# B&R Automation Studio project lab4
Automation Studio 4.5.2.102

## Configuration Real

### Hardware
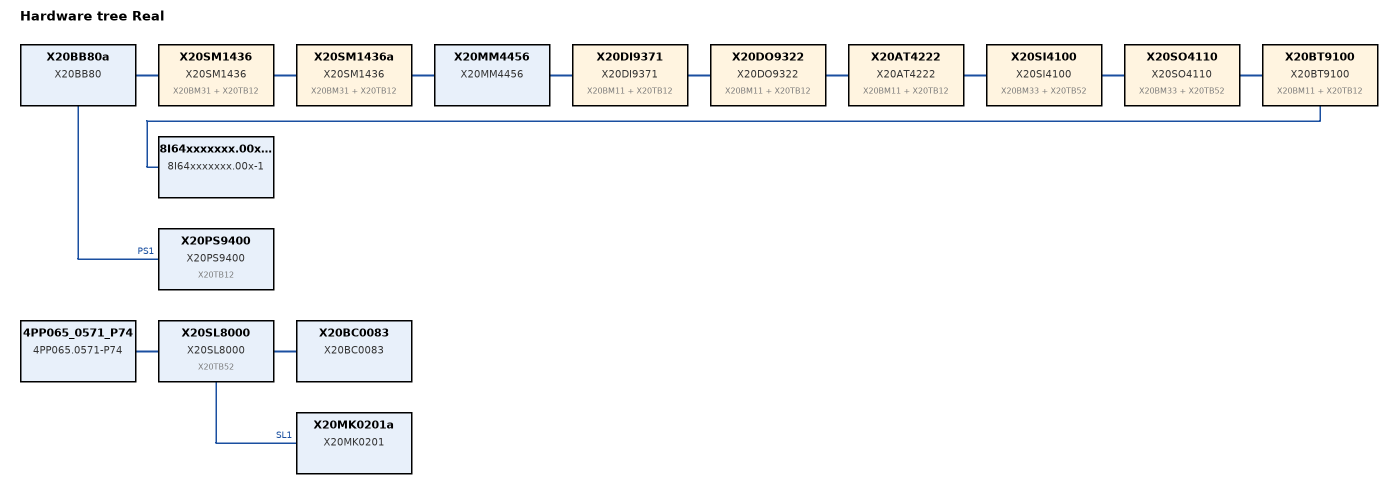
```
4PP065_0571_P74 : 4PP065.0571-P74 v1.1.2.0
  Connector IF5:
    ActivateDevice = 1
    Mode = Manual
    InternetAddress = 10.0.1.10
    SubnetMask = 255.255.255.0
  ConfigurationID = LabBR
  TimerDeviceType = EPLX2X
  TimerDevice = 4PP065_0571_P74.IF4
  TaskClassIdleTime = 2000
  Cyclic1Duration = 2000
  Cyclic1Tolerance = 0
  Cyclic1Output = 1
  Cyclic3Tolerance = 0
  VcObjectName = Visu
8I64xxxxxxx.00x-1 : 8I64xxxxxxx.00x-1 v1.3.9.1  [X2X1 -> X20BT9100.X2X1 [Cable Type=X2XCable, Length=10, Version=1.0.0.2]]
  BothEndSwitchesAreNormallyOpen_r1 = on
  QuickStopIsNormallyOpen_r1 = on
X20AT4222 : X20AT4222 v1.2.3.0  [SS1 -> X20TB12f.SS; SL -> X20BM11c.SL1]
X20BB80a : X20BB80 v1.0.2.0
X20BC0083 : X20BC0083 v2.7.0.0  [PLK1 -> X20SL8000.PLK2 (NodeNumber=2) [Cable Type=PowerlinkCable, Length=10, Version=1.0.0.2]; SL -> X20BB80a.SL1]
X20BM11a : X20BM11 v1.0.0.1  [X2X1 -> X20MM4456.X2X2]
X20BM11b : X20BM11 v1.0.0.1  [X2X1 -> X20BM11a.X2X2]
X20BM11c : X20BM11 v1.0.0.1  [X2X1 -> X20BM11b.X2X2]
X20BM11d : X20BM11 v1.0.0.1  [X2X1 -> X20BM33b.X2X2]
X20BM31a : X20BM31 v1.0.0.1  [X2X1 -> X20BB80a.IF1]
X20BM31b : X20BM31 v1.0.0.1  [X2X1 -> X20BM31a.X2X2]
X20BM33a : X20BM33 v1.0.0.4  [X2X1 -> X20BM11c.X2X2]
X20BM33b : X20BM33 v1.0.0.4  [X2X1 -> X20BM33a.X2X2]
X20BT9100 : X20BT9100 v1.0.3.0  [SS1 -> X20TB12g.SS; SL -> X20BM11d.SL1]
X20DI9371 : X20DI9371 v1.0.2.0  [SS1 -> X20TB12d.SS; SL -> X20BM11a.SL1]
X20DO9322 : X20DO9322 v1.0.3.0  [SS1 -> X20TB12e.SS; SL -> X20BM11b.SL1]
X20MK0201a : X20MK0201 v1.0.0.0  [SL -> X20SL8000.SL1]
X20MM4456 : X20MM4456 v1.1.5.0  [X2X1 -> X20BM31b.X2X2]
X20PS9400 : X20PS9400 v1.0.2.4  [SS1 -> X20TB12b.SS; PS -> X20BB80a.PS1]
X20SI4100 : X20SI4100 v1.10.1.1  [SS1 -> X20TB52b.SS; SL -> X20BM33a.SL1]
X20SL8000 : X20SL8000 v1.6.5.1  [PLK1 -> 4PP065_0571_P74.IF4 (NodeNumber=1) [Cable Type=PowerlinkCable, Length=10, Version=1.0.0.2]; PLK2 -> X20BC0083.PLK1 (NodeNumber=1) [Cable Type=PowerlinkCable, Length=10, Version=1.0.0.2]; SS1 -> X20TB52a.SS]
  SafeProject = SafeLOGIC-1
X20SM1436 : X20SM1436 v1.4.2.1  [SS1 -> X20TB12a.SS; SL -> X20BM31a.SL1]
X20SM1436a : X20SM1436 v1.4.2.1  [SS1 -> X20TB12c.SS; SL -> X20BM31b.SL1]
X20SO4110 : X20SO4110 v1.10.1.1  [SS1 -> X20TB52c.SS; SL -> X20BM33b.SL1]
  SafeLogicID = 2
  SafeModuleID = 3
X20TB12a : X20TB12 v1.0.0.0
X20TB12b : X20TB12 v1.0.0.0
X20TB12c : X20TB12 v1.0.0.0
X20TB12d : X20TB12 v1.0.0.0
X20TB12e : X20TB12 v1.0.0.0
X20TB12f : X20TB12 v1.0.0.0
X20TB12g : X20TB12 v1.0.0.0
X20TB52a : X20TB52 v1.0.0.1
X20TB52b : X20TB52 v1.0.0.1
X20TB52c : X20TB52 v1.0.0.1
```

### IoMap.iom - 4PP065_0571_P74/IoMap.iom
```iecst
VAR_CONFIG
	::SDCAxisCt2:posEnable.enable AT %IX."X20DI9371".DigitalInput04; (*Insert your comment here...*)
	::SDCAxisCt2:posEnableRight.enable AT %IX."X20DI9371".DigitalInput05; (*Insert your comment here...*)
	::SDCAxisCt1:posEnable.enable AT %IX."X20DI9371".DigitalInput04; (*Insert your comment here...*)
	::SDCAxisCt1:posEnableRight.enable AT %IX."X20DI9371".DigitalInput05; (*Insert your comment here...*)
	::SDCAxisCtr:posEnable.enable AT %IX."X20DI9371".DigitalInput02; (*Insert your comment here...*)
	::SDCAxisCtr:posEnableRight.enable AT %IX."X20DI9371".DigitalInput03; (*Insert your comment here...*)
	Cyclic#1.gAxis03_DrvIf.iLifeCnt AT %IB."8I64xxxxxxx.00x-1".SDC_LifeCnt;
	Cyclic#1.gAxis03_DrvIf.iDrvOK AT %IX."8I64xxxxxxx.00x-1".ETAD_Input_Bool_02;
	Cyclic#1.gAxis03_DrvIf.oSetTime AT %QW."8I64xxxxxxx.00x-1".SDC_SetTime;
	Cyclic#1.gAxis03_DrvIf.oSetPos AT %QW."8I64xxxxxxx.00x-1".LFRD_Output;
	Cyclic#1.gAxis03_DiDoIf.iLifeCntDriveReady AT %IB."8I64xxxxxxx.00x-1".SDC_LifeCnt;
	Cyclic#1.gAxis03_DiDoIf.iLifeCntDriveEnable AT %IB."8I64xxxxxxx.00x-1".SDC_LifeCnt;
	Cyclic#1.gAxis03_DiDoIf.oDriveEnable AT %QX."8I64xxxxxxx.00x-1".CMDD_Output_Bool_00;
	Cyclic#1.gAxis03_ModuleOk AT %QX."8I64xxxxxxx.00x-1".CMDD_Output_Bool_01;
	Cyclic#1.gAxis03_ModuleOk AT %QX."8I64xxxxxxx.00x-1".CMDD_Output_Bool_02;
	Cyclic#1.gAxis03_ModuleOk AT %IX."8I64xxxxxxx.00x-1".ModuleOk;
	Cyclic#1.gAxis03_DiDoIf.oDriveEnable AT %QX."8I64xxxxxxx.00x-1".CMDD_Output_Bool_03;
	Cyclic#1.gAxis03_DiDoIf.iDriveReady AT %IX."8I64xxxxxxx.00x-1".ETAD_Input_Bool_02;
	::SDCAxisCtr:pwm_period AT %QW."X20MM4456".PeriodDurationPWM;
	::SDCAxisCtr:coil_pwm_value AT %QW."X20MM4456".PulseWidthCurrentPWM04;
	::SDCAxisCtr:axis_X.pwm_value AT %QW."X20MM4456".PulseWidthCurrentPWM01;
	::SDCAxisCtr:axis_X.reset_error AT %QX."X20MM4456".ClearError01;
	::SDCAxisCtr:axis_X.reset_counter AT %QX."X20MM4456".ResetCounter01;
	::SDCAxisCtr:axis_X.counter AT %IW."X20MM4456".Counter01;
	::SDCAxisCtr:axis_X.endswitch_a_reached AT %IX."X20MM4456".StatusInput03; (*Logical condition input 01=Motor 01:A*)
	::SDCAxisCtr:axis_X.endswitch_b_reached AT %IX."X20MM4456".StatusInput04; (*Logical condition input 02=Motor 01:B*)
	::SDCAxisCtr:coil_powered AT %IX."X20DI9371".DigitalInput01;
	::SDCAxisCt1:axis_Y.pwm_value AT %QW."X20MM4456".PulseWidthCurrentPWM02;
	::SDCAxisCt1:axis_Y.reset_error AT %QX."X20MM4456".ClearError02;
	::SDCAxisCt1:axis_Y.reset_counter AT %QX."X20MM4456".ResetCounter02;
	::SDCAxisCt1:axis_Y.counter AT %IW."X20MM4456".Counter02;
	::SDCAxisCt1:axis_Y.endswitch_a_reached AT %IX."X20MM4456".StatusInput07;
	::SDCAxisCt1:axis_Y.endswitch_b_reached AT %IX."X20MM4456".StatusInput08;
	::SDCAxisCt2:axis_Z.pwm_value AT %QW."X20MM4456".PulseWidthCurrentPWM03;
	::SDCAxisCt2:axis_Z.reset_error AT %QX."X20MM4456".ClearError03;
	::SDCAxisCt2:axis_Z.reset_counter AT %QX."X20MM4456".ResetCounter03;
	::SDCAxisCt2:axis_Z.counter AT %IW."X20MM4456".Counter03;
	::SDCAxisCt2:axis_Z.endswitch_a_reached AT %IX."X20MM4456".StatusInput11;
	::SDCAxisCt2:axis_Z.endswitch_b_reached AT %IX."X20MM4456".StatusInput12;
	::SDCAxisCt1:coil_powered AT %IX."X20DI9371".DigitalInput02;
	::SDCAxisCt2:coil_powered AT %IX."X20DI9371".DigitalInput03;
END_VAR
```

### Acp10map1.ncm - 4PP065_0571_P74/Motion/Acp10map1.ncm
```
NcMapping (NcSwId=ACP10, DisabledNodesAreHidden=False)
  NcObject AxisX (ModuleAddress=SDC_IF1.ST2, InterfaceType=SDC, Type=ncAXIS, Channel=1, AcoposSimulation=Off, InitParameter=AxisInit, AcoposParameter=AxisApt, AdditionalData=CNC_Enabled="1" , Disabled=FALSE, ModuleDisabled=FALSE)
  NcObject AxisY (ModuleAddress=SDC_IF1.ST3, InterfaceType=SDC, Type=ncAXIS, Channel=1, AcoposSimulation=Off, InitParameter=AxisInit, AcoposParameter=AxisApt, AdditionalData=CNC_Enabled="1" , Disabled=FALSE)
  NcObject AxisZ (ModuleAddress=SDC_IF1.ST4, InterfaceType=SDC, Type=ncAXIS, Channel=1, AcoposSimulation=Off, InitParameter=AxisInit, AcoposParameter=AxisApt, AdditionalData=CNC_Enabled="1" , Disabled=FALSE)
```

## Logical view

### Package Logical/Libraries - Global libraries

### Library Logical/Libraries/Library (ANSIC)

#### Library.fun
```iecst
FUNCTION_BLOCK FB_Motor (*TODO: Add your comment here*) (*$GROUP=User,$CAT=User,$GROUPICON=User.png,$CATICON=User.png*)
	VAR_INPUT
		in : REAL;
	END_VAR
	VAR_OUTPUT
		out_w : REAL;
		out_phi : REAL;
	END_VAR
	VAR
		k_e : REAL;
		T_m : REAL;
		dt : REAL;
		integrator : FB_Integrator;
		integrator_phi : FB_Integrator;
	END_VAR
END_FUNCTION_BLOCK

FUNCTION_BLOCK FB_Integrator (*TODO: Add your comment here*) (*$GROUP=User,$CAT=User,$GROUPICON=User.png,$CATICON=User.png*)
	VAR_INPUT
		in : REAL;
		dt : REAL;
	END_VAR
	VAR_OUTPUT
		out : REAL;
	END_VAR
	VAR
		state : REAL := 0.0;
	END_VAR
END_FUNCTION_BLOCK

FUNCTION_BLOCK FB_Controller (* *) (*$GROUP=User,$CAT=User,$GROUPICON=User.png,$CATICON=User.png*)
	VAR_INPUT
		in : REAL;
	END_VAR
	VAR_OUTPUT
		out : REAL;
	END_VAR
	VAR
		k_i : REAL;
		sum : REAL;
		k_p : REAL;
		dt : REAL;
		max_abs_value : REAL;
		integrator : FB_Integrator;
		last_sum : REAL;
	END_VAR
END_FUNCTION_BLOCK

FUNCTION_BLOCK FB_Endswitch (*TODO: Add your comment here*) (*$GROUP=User,$CAT=User,$GROUPICON=User.png,$CATICON=User.png*)
	VAR_INPUT
		in : REAL;
		neg_value : REAL;
		pos_value : REAL;
	END_VAR
	VAR_OUTPUT
		neg_reached : BOOL;
		pos_reached : BOOL;
	END_VAR
END_FUNCTION_BLOCK

FUNCTION_BLOCK FB_Axis (*TODO: Add your comment here*) (*$GROUP=User,$CAT=User,$GROUPICON=User.png,$CATICON=User.png*)
	VAR_INPUT
		reset_error : BOOL;
		endswitch_a_reached : BOOL;
		endswitch_b_reached : BOOL;
		pwm_percentage : SINT;
	END_VAR
	VAR_OUTPUT
		reset_counter : BOOL;
		pwm_value : INT;
	END_VAR
	VAR_OUTPUT RETAIN
		counter : INT;
	END_VAR
	VAR_OUTPUT
		speed : REAL;
	END_VAR
	VAR
		last_counter : INT;
	END_VAR
END_FUNCTION_BLOCK

{REDUND_ERROR} FUNCTION_BLOCK Pos (*TODO: Add your comment here*) (*$GROUP=User,$CAT=User,$GROUPICON=User.png,$CATICON=User.png*)
	VAR_INPUT
		enable : BOOL;
	END_VAR
END_FUNCTION_BLOCK
```

#### Pos.c
```c
#include <bur/plctypes.h>
#ifdef __cplusplus
	extern "C"
	{
#endif
	#include "Library.h"
#ifdef __cplusplus
	};
#endif
/* TODO: Add your comment here */
void Pos(struct Pos* inst)
{
	/*TODO: Add your code here*/
}
```

### Data object Logical/AxisInit (Ax)

#### AxInitAcp10.ax
```
InitParameter (Version=5.2.1, NcSwId=ACP10)
  ACP10AXIS_typ:
    dig_in:
      level:
        reference = ncACTIV_HI
        pos_hw_end = ncACTIV_HI
        neg_hw_end = ncACTIV_HI
        trigger1 = ncACTIV_HI
        trigger2 = ncACTIV_HI
    encoder_if:
      parameter:
        count_dir = ncSTANDARD
        scaling:
          load:
            units = 3000
            rev_motor = 1
    limit:
      parameter:
        v_pos = 7500.0
        v_neg = 7500.0
        a1_pos = 10000.0
        a2_pos = 10000.0
        a1_neg = 10000.0
        a2_neg = 10000.0
        t_jolt = 0.0
        t_in_pos = 0.0
        pos_sw_end = 8388607
        neg_sw_end = -8388608
        ds_warning = 500.0
        ds_stop = 1000.0
        a_stop = 1.0E+30
        dv_stop = 0.0
        dv_stop_mode = ncOFF
    controller:
      mode = ncPOSITION
      position:
        kv = 10.0
        tn = 0.0
        t_predict = 0.04
        t_total = 0.04
        p_max = 10000.0
        i_max = 0.0
      speed:
        kv = 2.0
        tn = 0.0
        t_filter = 0.0
        isq_filter1:
          type = ncOFF
          a0 = 0.0
          a1 = 0.0
          b0 = 0.0
          b1 = 0.0
          b2 = 0.0
          c0_par_id = 0
          c1_par_id = 0
        isq_filter2:
          type = ncOFF
          a0 = 0.0
          a1 = 0.0
          b0 = 0.0
          b1 = 0.0
          b2 = 0.0
          c0_par_id = 0
          c1_par_id = 0
        isq_filter3:
          type = ncOFF
          a0 = 0.0
          a1 = 0.0
          b0 = 0.0
          b1 = 0.0
          b2 = 0.0
          c0_par_id = 0
          c1_par_id = 0
      uf:
        type = ncLINEAR
        auto_config = ncMOTOR_PAR
        u0 = 0.0
        un = 0.0
        fn = 50.0
        k_f_slip = 0.0
      ff:
        torque_load = 0.0
        torque_pos = 0.0
        torque_neg = 0.0
        kv_torque = 0.0
        inertia = 0.0
        t_filter_a = 0.0
    move:
      stop:
        parameter[0]:
          decel_ramp = ncA_LIMIT
          controller = ncON
        parameter[1]:
          decel_ramp = ncA_LIMIT
          controller = ncON
        parameter[2]:
          decel_ramp = ncA_LIMIT
          controller = ncON
        parameter[3]:
          decel_ramp = ncA_LIMIT
          controller = ncON
        quickstop:
          decel_ramp = ncA_LIMIT
          t_jolt = 0.0
        drive_error:
          decel_ramp = ncA_LIMIT
      homing:
        parameter:
          s = 0
          v_switch = 6000.0
          v_trigger = 2000.0
          a = 10000.0
          mode = ncDIRECT
          edge_sw = ncNEGATIVE
          start_dir = ncPOSITIVE
          trigg_dir = ncNEGATIVE
          ref_pulse = ncOFF
          fix_dir = ncOFF
          tr_s_block = 0.0
          torque_lim = 0.0
          ds_block = 0.0
          ds_stop = 0.0
      basis:
        parameter:
          v_pos = 4000.0
          v_neg = 4000.0
          a1_pos = 10000.0
          a2_pos = 10000.0
          a1_neg = 10000.0
          a2_neg = 10000.0
    message:
      text:
        parameter:
          format = ncBREAK
          columns = 80
          data_modul
```

### Data object Logical/CncInit (Cns)

- CncInit.cns (not shown)

### Program Logical/SDCAxisCtrl_X (ANSIC)

#### Variables.var
```iecst
VAR
	min_task : INT := 7000;
	desired_speed : INT := 0;
	axis_X : FB_Axis;
	coil_powered : BOOL := FALSE;
	coil_pwm_value : {REDUND_UNREPLICABLE} INT := 200;
	fb_controller : FB_Controller;
	pwm_period : {REDUND_UNREPLICABLE} UINT := 200;
	posEnable : Pos := (0);
	posEnableRight : Pos := (0);
END_VAR
```

#### Main.c
```c
#include <bur/plctypes.h>

#ifdef _DEFAULT_INCLUDES
	#include <AsDefault.h>
#endif

void increase_counters(void);

void _INIT ProgramInit(void)
{
	AxisX_HW.EncIf1_Typ = ncSDC_ENC16;
	AxisX_HW.DiDoIf_Typ = ncSDC_DIDO;
	AxisX_HW.DrvIf_Typ = ncSDC_DRVSERVO16;

	strcpy(AxisX_HW.EncIf1_Name, "AxisX_EncIf");
	strcpy(AxisX_HW.DrvIf_Name, "AxisX_DrvIf");
	strcpy(AxisX_HW.DiDoIf_Name, "AxisX_DiDoIf");

	AxisX_EncIf.iEncOK = 1;
	AxisX_DrvIf.iDrvOK = 1;
	AxisX_DrvIf.iStatusEnable = 1;
	AxisX_DiDoIf.iDriveReady = 1;

	fb_controller.dt = 0.002;
	fb_controller.k_i = 0.16;
	fb_controller.k_p = 0.0064;
	fb_controller.max_abs_value = 24.0;

	pwm_period = 200;
}

void _CYCLIC ProgramCyclic(void)
{
	if (posEnable.enable) {
		//	axis_X.endswitch_a_reached = 1;
		AxisX_DrvIf.oSetPos = -10000;
	} else if (posEnableRight.enable) {
		AxisX_DrvIf.oSetPos = 10000;
	}
	FB_Axis(&axis_X);
	coil_pwm_value = coil_powered ? 32767 : 0;

	increase_counters();

	AxisX_EncIf.iActTime = (INT)	AsIOTimeCyclicStart();
	AxisX_EncIf.iActPos = axis_X.counter;
	AxisX_DiDoIf.iPosHwEnd = axis_X.endswitch_b_reached;
	AxisX_DiDoIf.iNegHwEnd = axis_X.endswitch_a_reached;
	fb_controller.in = AxisX_DrvIf.oSetPos;

	if((fb_controller.in<min_task)&&(fb_controller.in>(-min_task))) fb_controller.in = 0;
	fb_controller.in = fb_controller.in * 6500/32767 - axis_X.speed;

	FB_Controller(&fb_controller);

	axis_X.pwm_value = fb_controller.out / 24.0 * 32767;
}

void increase_counters(void)
{
	AxisX_EncIf.iLifeCnt++;
	AxisX_DiDoIf.iLifeCntDriveEnable++;
	AxisX_DiDoIf.iLifeCntDriveReady++;
	AxisX_DiDoIf.iLifeCntNegHwEnd++;
	AxisX_DiDoIf.iLifeCntPosHwEnd++;
	AxisX_DiDoIf.iLifeCntReference++;
	AxisX_DrvIf.iLifeCnt++;
}

void _EXIT ProgramExit(void)
{
	// Insert code here

}
```

### Program Logical/SDCAxisCtrl_Y (ANSIC)

#### Variables.var
```iecst
VAR
	min_task : INT := 7000;
	desired_speed : INT := 0;
	axis_Y : FB_Axis;
	coil_powered : BOOL := FALSE;
	coil_pwm_value : {REDUND_UNREPLICABLE} INT := 200;
	fb_controller : FB_Controller;
	pwm_period : {REDUND_UNREPLICABLE} UINT := 200;
	posEnable : Pos := (0);
	posEnableRight : Pos := (0);
END_VAR
```

#### Main.c
```c
#include <bur/plctypes.h>

#ifdef _DEFAULT_INCLUDES
	#include <AsDefault.h>
#endif

void _INIT ProgramInit(void)
{
	AxisY_HW.EncIf1_Typ = ncSDC_ENC16;
	AxisY_HW.DiDoIf_Typ = ncSDC_DIDO;
	AxisY_HW.DrvIf_Typ = ncSDC_DRVSERVO16;

	strcpy(AxisY_HW.EncIf1_Name, "AxisY_EncIf");
	strcpy(AxisY_HW.DrvIf_Name, "AxisY_DrvIf");
	strcpy(AxisY_HW.DiDoIf_Name, "AxisY_DiDoIf");

	AxisY_EncIf.iEncOK = 1;
	AxisY_DrvIf.iDrvOK = 1;
	AxisY_DrvIf.iStatusEnable = 1;
	AxisY_DiDoIf.iDriveReady = 1;

	fb_controller.dt = 0.002;
	fb_controller.k_i = 0.16;
	fb_controller.k_p = 0.0064;
	fb_controller.max_abs_value = 24.0;

	pwm_period = 200;

}

void _CYCLIC ProgramCyclic(void)
{
	if (posEnable.enable) {
		//	axis_X.endswitch_a_reached = 1;
		AxisY_DrvIf.oSetPos = -10000;
	} else if (posEnableRight.enable) {
		AxisY_DrvIf.oSetPos = 10000;
	}
	FB_Axis(&axis_Y);
	coil_pwm_value = coil_powered ? 32767 : 0;

	increase_counters();

	AxisY_EncIf.iActTime = (INT)	AsIOTimeCyclicStart();
	AxisY_EncIf.iActPos = axis_Y.counter;
	AxisY_DiDoIf.iPosHwEnd = axis_Y.endswitch_b_reached;
	AxisY_DiDoIf.iNegHwEnd = axis_Y.endswitch_a_reached;
	fb_controller.in = AxisY_DrvIf.oSetPos;

	if((fb_controller.in<min_task)&&(fb_controller.in>(-min_task))) fb_controller.in = 0;
	fb_controller.in = fb_controller.in * 6500/32767 - axis_Y.speed;

	FB_Controller(&fb_controller);

	axis_Y.pwm_value = fb_controller.out / 24.0 * 32767;
}

void increase_counters(void)
{
	AxisY_EncIf.iLifeCnt++;
	AxisY_DiDoIf.iLifeCntDriveEnable++;
	AxisY_DiDoIf.iLifeCntDriveReady++;
	AxisY_DiDoIf.iLifeCntNegHwEnd++;
	AxisY_DiDoIf.iLifeCntPosHwEnd++;
	AxisY_DiDoIf.iLifeCntReference++;
	AxisY_DrvIf.iLifeCnt++;
}

void _EXIT ProgramExit(void)
{
	// Insert code here

}
```

### Program Logical/SDCAxisCtrl_Z (ANSIC)

#### Variables.var
```iecst
VAR
	min_task : INT := 7000;
	desired_speed : INT := 0;
	axis_Z : FB_Axis;
	coil_powered : BOOL := FALSE;
	coil_pwm_value : {REDUND_UNREPLICABLE} INT := 200;
	fb_controller : FB_Controller;
	pwm_period : {REDUND_UNREPLICABLE} UINT := 200;
	posEnable : Pos := (0);
	posEnableRight : Pos := (0);
END_VAR
```

#### Main.c
```c
#include <bur/plctypes.h>

#ifdef _DEFAULT_INCLUDES
	#include <AsDefault.h>
#endif

void _INIT ProgramInit(void) {

	AxisZ_HW.EncIf1_Typ = ncSDC_ENC16;
	AxisZ_HW.DiDoIf_Typ = ncSDC_DIDO;
	AxisZ_HW.DrvIf_Typ = ncSDC_DRVSERVO16;

	strcpy(AxisZ_HW.EncIf1_Name, "AxisZ_EncIf");
	strcpy(AxisZ_HW.DrvIf_Name, "AxisZ_DrvIf");
	strcpy(AxisZ_HW.DiDoIf_Name, "AxisZ_DiDoIf");

	AxisZ_EncIf.iEncOK = 1;
	AxisZ_DrvIf.iDrvOK = 1;
	AxisZ_DrvIf.iStatusEnable = 1;
	AxisZ_DiDoIf.iDriveReady = 1;

	fb_controller.dt = 0.002;
	fb_controller.k_i = 0.16;
	fb_controller.k_p = 0.0064;
	fb_controller.max_abs_value = 24.0;

	pwm_period = 200;
}

void _CYCLIC ProgramCyclic(void)
{
	if (posEnable.enable) {
		//	axis_X.endswitch_a_reached = 1;
		AxisZ_DrvIf.oSetPos = -10000;
	} else if (posEnableRight.enable) {
		AxisZ_DrvIf.oSetPos = 10000;
	}
	FB_Axis(&axis_Z);
	coil_pwm_value = coil_powered ? 32767 : 0;

	increase_counters();

	AxisZ_EncIf.iActTime = (INT)	AsIOTimeCyclicStart();
	AxisZ_EncIf.iActPos = axis_Z.counter;
	AxisZ_DiDoIf.iPosHwEnd = axis_Z.endswitch_b_reached;
	AxisZ_DiDoIf.iNegHwEnd = axis_Z.endswitch_a_reached;
	fb_controller.in = AxisZ_DrvIf.oSetPos;

	if((fb_controller.in<min_task)&&(fb_controller.in>(-min_task))) fb_controller.in = 0;
	fb_controller.in = fb_controller.in * 6500/32767 - axis_Z.speed;

	FB_Controller(&fb_controller);

	axis_Z.pwm_value = fb_controller.out / 24.0 * 32767;

}

void increase_counters(void)
{
	AxisZ_EncIf.iLifeCnt++;
	AxisZ_DiDoIf.iLifeCntDriveEnable++;
	AxisZ_DiDoIf.iLifeCntDriveReady++;
	AxisZ_DiDoIf.iLifeCntNegHwEnd++;
	AxisZ_DiDoIf.iLifeCntPosHwEnd++;
	AxisZ_DiDoIf.iLifeCntReference++;
	AxisZ_DrvIf.iLifeCnt++;

}

void _EXIT ProgramExit(void)
{
	// Insert code here

}
```

Listed in the project but not available here: Logical/Global.typ, Logical/Global.var, Logical/Libraries/Library/FB_Motor.c, Logical/Libraries/Library/FB_Controller.c, Logical/Libraries/Library/FB_Integrator.c, Logical/Libraries/Library/FB_Endswitch.c, Logical/Libraries/Library/FB_Axis.c, Logical/AxisApt, Logical/Types.typ, Logical/acp10etxen, Logical/ncsdcctrl, Logical/gAxis03obj, Logical/GmcIpConfig, Logical/GmcIpUserConfig, Logical/CncProg1
